(* CoDeSys 2.3 export: SW_VERSION.EXP *)

(* POU Autocode/SW_Version, ST *)
PROGRAM SW_Version 
VAR 
	SW_Git_Commit_s32	: DINT;		(* First 7 characters of the current git commit, hex *) 
	SW_Git_Hash_as8	: STRING;	(* First 7 characters of the current git commit, hex *) 
END_VAR 
(*********************************************) 
(*  DON'T MAKE ANY CHANGES TO THIS PROGRAM!! *) 
(*     FILE WAS AUTOMATICALLY GENERATED!!    *) 
(*********************************************) 
SW_Git_Commit_s32 := 16#dceb9f2;
SW_Git_Hash_as8 := 'dceb9f2';
END_PROGRAM
